FUNCTION_BLOCK ServoMotor EXTENDS Motor
VAR_INPUT
END_VAR
VAR_OUTPUT
END_VAR
VAR
	position : INT;
END_VAR

METHOD turn90Deg
VAR_INPUT
END_VAR
position := 90;
END_METHOD

END_FUNCTION_BLOCK

(* stored: Version 1.1.0.1, ProductVersion 3.1.4024.11
   POU ServoMotor: Id {3ea56d1d-3e72-4965-be66-010de9455a87}, SpecialFunc None
   Method turn90Deg: Id {022882b8-d2a5-42ab-9b0e-22e69c185fc7} *)
